PROGRAM MAIN_S2

VAR
	b110SyncState AT %I* :UINT ;
	b110State AT %I* :UINT;  

	AktiveSystem : BOOL := TRUE;
	bSwitch : BOOL := FALSE;
	nState: UINT;
	CycelCount :ARRAY[1..GVL_MC.nNumMovers] OF INT;
	MoverState :ARRAY[1..GVL_MC.nNumMovers] OF UINT;
	nForCounter ,i: UINT;
	Velo : LREAL := 2000;


	ipXlMover : 	I_XtsXlMover1;


	state AT %Q* : INT := -1;
	arrivedOTCID : OTCID;
	Start :BOOL;
	bAlldone : BOOL;


	test : otcid; 
	XPU_Number : UINT := 1; 	
	
	Short : BOOL;
	
	XtsOutterLoopOid: OTCID ;	
	XtsShortcutOid: OTCID ;

	Init : BOOL ; 
	EndTrack : INT :=E_TrackNum.MainStart ;
 	StartTrack : INT :=E_TrackNum.MainStart ;
	MoverNo : DINT;
	SystemReady: BOOL;
	
	cmdFeedback: Tc3_XtsInterface.XtsCommandFeedback;
	BUFFER: BYTE;
	
	xEapStart AT %I*: BOOL;
	xEAPReset AT %I*: BOOL;
	EtherCATModulesWCState AT %I*: BOOL;
	EhterCATFault: BOOL;
	SyncFault: BOOL;
	
	temp: HRESULT;
	
	haltDynamics : DynamicConstraint_PathXY;
	stMoverConfigSlow	: ST_MoverConfig;
	stMoverConfigNormal : ST_MoverConfig;
	stMoverConfigFast  : ST_MoverConfig;
	stMoverCfgAggressive : ST_MoverConfig;
	stMoverCfgHalt : ST_MoverConfig;
	MoverStopDone : BOOL;
	Fault : BOOL;
	Fp_error : r_trig;
	AllDone : BOOL;
	InitDone  :BOOL;
END_VAR

// =====================
// Initalize XTS Utility
GVL_MC.fbXtsEnvironment.Init(GVL_MC.cmdFeedback);
IF NOT GVL_MC.cmdFeedback.IsDone THEN
	RETURN;
END_IF

IF  GVL_DataExchange.Dynamics.V = 0 THEN
	stMoverConfigNormal.Velo	:=	1000;
	stMoverConfigNormal.Accel	:=	4000;
	stMoverConfigNormal.Decel	:=	4000;
	stMoverConfigNormal.Jerk	:=	16000;
ELSE
	stMoverConfigNormal.Velo	:=	GVL_DataExchange.Dynamics.v;
	stMoverConfigNormal.Accel	:=	GVL_DataExchange.Dynamics.A;
	stMoverConfigNormal.Decel	:=	GVL_DataExchange.Dynamics.D;
	stMoverConfigNormal.Jerk	:=	GVL_DataExchange.Dynamics.J;
END_IF
// =====================
GVL_MC.ipXtsProcessingUnit :=  GVL_MC.fbXtsEnvironment.ProcessingUnit(XPU_Number,0);
AllDone := TRUE;
FOR i := 1 TO GVL_MC.nNumMovers DO 
	
	IF NOT InitDone  THEN
		ipXlMover  :=  GVL_MC.fbXtsEnvironment.ProcessingUnit(XPU_Number, 0).XlMover(i, 0);
		AllDone := AllDone AND GVL_MC.fbMover[i].Init(ipXlMover, GVL_MC.ipXtsProcessingUnit); 
	END_IF
	InitDone := alldone;
	
	Fp_error(clk := GVL_MC.fbMover[i].P_PlanarMover.Error AND GVL_MC.fbMover[i].XtsXlMover.GetIsActive(0) AND state = 100);
	IF Fp_error.Q THEN
		state := 140;
		Fault := TRUE;

		ADSLOGSTR(msgCtrlMask:= ADSLOG_MSGTYPE_LOG , msgFmtStr:= 'Mover %s Faulted ' , strArg:= INT_TO_STRING(i));
	ELSE
		Fault := FALSE;
	END_IF
	
	
	GVL_MC.Feedback[i].Update();
	GVL_MC.fbMover[i].CycleUpdate();
	GVL_MC.iMover[i] := GVL_MC.fbMover[i];
	GVL_MC.fbMover[i].P_Dynamics.SetValuesVADJ(stMoverConfigNormal.Velo,stMoverConfigNormal.Accel, stMoverConfigNormal.Decel, stMoverConfigNormal.Jerk);
	GVL_MC.fbMover[i].P_MoveOnTrackOptions.gap := 900;
	GVL_MC.fbMover[i].P_MoveOnTrackOptions.direction := MC_Direction.mcDirectionPositive;
	GVL_MC.fbMover[i].P_MoveOnTrackOptions.gapMode := MC_GAP_MODE_ON_TRACK.Fast1D;
	
	GVL_DataExchange.aMoverInfos[i] :=  GVL_MC.fbMover[i].P_MoverInfos;
END_FOR	

FOR i := 1 TO GVL_MC.nNumTracks DO 
	GVL_MC.aMcTracks[i].Update();
	GVL_MC.TrackFeedback[i].Update();
END_FOR	

IF NOT Init THEN
	Init := TRUE;
END_IF

IF state <99 AND xEAPReset THEN 
	state := 0; 
END_IF

IF state = 99 AND xEAPStart THEN 
	state := 100; 
END_IF

IF EtherCATModulesWCState THEN 
	EhterCATFault := TRUE;
END_IF  

IF b110SyncState <>1 THEN 
	SyncFault := TRUE; 
END_IF



CASE state OF
	0: 
		
		FOR i := 1 TO GVL_MC.nNumTracks DO  
			GVL_MC.aMcTracks[i].Enable(GVL_MC.TrackFeedback[i]);
			state := 1;
		END_FOR
		
	1: 	
		bAlldone := TRUE;
		FOR i := 1 TO GVL_MC.nNumTracks DO  
			bAlldone := bAlldone AND GVL_MC.aMcTracks[i].MCTOPLC_STD.State = MC_PLANAR_STATE.Enabled ;
		END_FOR
			
 		IF bAlldone THEN
			state := 2;
		END_IF

	2:	
		FOR i := 1+GVL_MC.nNumActiveMovers TO GVL_MC.nNumMovers DO  
			GVL_MC.fbMover[i].XlProcessingUnit.XlMover(i,0).SetStartupTrackPosition(0.2,0);	
			GVL_MC.fbMover[i].XlProcessingUnit.XlMover(i,0).SetIsVirtualFeedbackEnabled(1,0);
			GVL_MC.fbMover[i].XlProcessingUnit.XlMover(i,0).TriggerArrive(0);
		END_FOR
		IF  GVL_MC.nNumActiveMovers > 0 THEN
			FOR i :=1  TO GVL_MC.nNumActiveMovers DO 	
				GVL_MC.fbMover[i].XlProcessingUnit.XlMover(i,0).SetIsVirtualFeedbackEnabled(0,0);
			END_FOR 
		END_IF			
		state := 3;
		
	3:
		FOR i := 1 TO GVL_MC.fbXtsEnvironment.ProcessingUnit(1, 0).XlPartCount() DO
			 GVL_MC.fbXtsEnvironment.ProcessingUnit(1, 0).XlPart(i, 0).TriggerReset(0);
		END_FOR
		
		state := 5;
		
	5: 

		
		IF AktiveSystem THEN
			state := 10;
		ELSE
			state := 100;
		END_IF	

	10:
		FOR i := 1 TO GVL_MC.nNumActiveMovers DO
			GVL_MC.fbMover[i].P_PlanarMover.Reset(0);
		END_FOR
		state := 11;
 	11:
		FOR i := 1 TO GVL_MC.nNumActiveMovers DO	
			GVL_MC.fbMover[i].P_PlanarMover.Enable(0);		
		END_FOR
		state := 15;	
	15:
		bAlldone := TRUE;
		FOR i := 1 TO GVL_MC.nNumActiveMovers DO  
			bAlldone := bAlldone AND GVL_MC.fbMover[i].P_PlanarMover.MCTOPLC.STD.State = MC_PLANAR_STATE.Enabled;	
		END_FOR
		
		IF bAlldone THEN
			state := 18;
		END_IF
	18: 
	
		FOR i := 1 TO GVL_MC.nNumActiveMovers DO  
			GVL_MC.fbMover[i].JoinNearestTrack(aMcTracks,nNumTracks );	
		END_FOR
		state := 20;
	
	20:
		bAlldone := TRUE;
		FOR i := 1 TO GVL_MC.nNumActiveMovers DO
			bAlldone := bAlldone AND GVL_MC.fbMover[i].fbPlanarMover.MCTOPLC.STD.CommandMode = MC_PLANAR_MOVER_COMMAND_MODE.OnTrack  ;	
			MoverState[i] := 10;
			
		END_FOR

		IF bAlldone THEN
			state := 99;
		END_IF
		
	100: 
		arrivedOTCID := GVL_MC.EnterSystem.PopFirstMoverInQueue();
		IF arrivedOTCID <> 0 THEN
			FOR i := 1  TO GVL_MC.nNumMovers DO
				IF GVL_MC.fbMover[i].p_MoverOTCID = arrivedOTCID THEN
					MoverState[i] := 0;
				END_IF
			END_FOR
		END_IF
	
		FOR i := 1 TO GVL_MC.nNumMovers DO 
			CASE MoverState[i] OF 
		
			0:
				IF MoverNo <> 0 AND_THEN GVL_MC.fbMover[MoverNo].P_PlanarMover.MCTOPLC.SETONTRACK.TrackOID =  GVL_MC.aMcTracks[E_TrackNum.MainStart].MCTOPLC_STD.TrackOID THEN
					Short := FALSE;
				END_IF
		
				IF GVL_MC.fbMover[i].P_PlanarMover.MCTOPLC.SETONTRACK.SetPos > 100  THEN
					IF NOT short AND bSwitch  THEN
						GVL_MC.fbMover[i].MoveOnTrack(GVL_MC.aMcTracks[E_TrackNum.MainStart],GVL_MC.aMcTracks[E_TrackNum.MainStart].GetLength()/2,GVL_MC.defaultGap);
						MoverNo := i;
						Short := TRUE;
						MoverState[i] := 10;
					ELSE
						GVL_MC.fbMover[i].MoveOnTrack(GVL_MC.aMcTracks[EndTrack],GVL_MC.aMcTracks[EndTrack].GetLength()/2,GVL_MC.defaultGap);			
						MoverState[i] := 10;
					END_IF				
				END_IF
								
			10:
				IF(  GVL_MC.fbMover[i].P_PlanarMover.MCTOPLC.SETONTRACK.SetPos > 500 AND GVL_MC.fbMover[i].P_PlanarMover.MCTOPLC.SETONTRACK.TrackOID <>  GVL_MC.aMcTracks[StartTrack].MCTOPLC_STD.TrackOID) OR GVL_MC.nNumTracks =1 THEN
					GVL_MC.fbMover[i].MoveOnTrack(GVL_MC.aMcTracks[EndTrack],GVL_MC.aMcTracks[EndTrack].GetLength() - 1500,GVL_MC.defaultGap) ;//VElo*0.35);
					MoverState[i] := 11;
				END_IF
			11:	
				//special command no chance to break in time 
				IF  SystemReady  THEN
					GVL_MC.fbMover[i].MoveOnTrack(GVL_MC.aMcTracks[EndTrack],GVL_MC.aMcTracks[EndTrack].GetLength() - 200,GVL_MC.defaultGap);
					//GVL_MC.fbMover[i].MoveOnTrack(GVL_MC.aMcTracks[EndTrack],GVL_MC.aMcTracks[EndTrack].GetLength()-200);
					MoverState[i] := 12;
				END_IF		
			12: IF GVL_MC.fbMover[i].P_PlanarMover.MCTOPLC.SETONTRACK.SetPos > GVL_MC.aMcTracks[EndTrack].GetLength() - 2300 AND 
				(GVL_MC.fbMover[i].P_PlanarMover.MCTOPLC.SETONTRACK.TrackOID = GVL_MC.aMcTracks[EndTrack].MCTOPLC_STD.TrackOID) AND SystemReady THEN 
					GVL_MC.fbMover[i].LeaveSystemAt(GVL_MC.ExitSystem, GVL_MC.defaultGap); 
					MoverState[i] := 15; 
				END_IF	
				
			15:
			 	IF GVL_MC.fbMover[i].XlProcessingUnit.XlMover(i,0).GetIsVirtualFeedbackEnabled(0) AND //In some cases the planar mover gots an error, we have to evaluate why
					GVL_MC.fbMover[i].P_PlanarMover.Error THEN
					GVL_MC.fbMover[i].P_PlanarMover.Reset(0);
					MoverState[i] := 16; 
				END_IF
				
			16: 
				GVL_MC.fbMover[i].P_PlanarMover.Disable(0);
				MoverState[i] := 17; 
			END_CASE
		END_FOR
		
		140:
			FOR i := 1 TO GVL_MC.nNumMovers DO  
				GVL_MC.fbMover[i].P_PlanarMover.Halt(GVL_MC.Feedback[i], haltDynamics);
			END_FOR	
			
				state := 145;
			
		145:
			bAllDone := TRUE;
				FOR i := 1 TO GVL_MC.nNumMovers DO  
				IF NOT(GVL_MC.Feedback[i].Done OR GVL_MC.Feedback[i].Error) THEN
					bAllDone := FALSE;
					EXIT;
				END_IF
			END_FOR
			
			IF bAllDone THEN
				state := 150;
			END_IF
		
		//Disable
		150:
			MoverStopDone := TRUE;
			FOR i := 1 TO GVL_MC.nNumMovers DO  
					GVL_MC.fbMover[i].P_PlanarMover.Disable(GVL_MC.Feedback[i]);
			END_FOR
				
			state := 0;
		
	
END_CASE

END_PROGRAM

(* stored: Version 1.1.0.1, ProductVersion 3.1.4026.11
   POU MAIN_S2: Id {eb537839-0cb8-4f4d-83cf-5c0c733fdb11}, SpecialFunc None *)
